(* CoDeSys 2.3.9.42 project: Revers privod_96.pro *)
(* Libraries: STANDARD.LIB 4.10.05 11:14:46, IECSFC.LIB 13.4.06 15:51:28, ANALYZATION.LIB 5.10.99 09:05:06 *)

(* Global variable list: Global_Variables *)
VAR_GLOBAL
	KM1, KM2:BOOL;
END_VAR

(* POU PLC_PRG, ST *)
PROGRAM PLC_PRG
VAR
	posy: INT;
END_VAR
Control();
Puskatel();

IF KM1 THEN
posy:=posy-1;
END_IF

IF KM2 THEN
posy:=posy+1;
END_IF
END_PROGRAM

(* POU Control, LD *)
PROGRAM Control
VAR
	S0: BOOL;
	SI: BOOL;
	SD: BOOL;
END_VAR
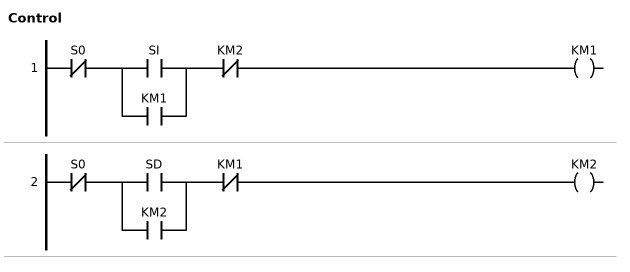
_LD_ (* Ladder Diagram *)
NETWORK 1
	[/S0] - { [SI] | [KM1] } - [/KM2] --- (KM1)
NETWORK 2
	[/S0] - { [SD] | [KM2] } - [/KM1] --- (KM2)
_END_LD_
(* the same logic as Structured Text *)
(* Network 1 *)
KM1 := NOT S0 AND (SI OR KM1) AND NOT KM2;
(* Network 2 *)
KM2 := NOT S0 AND (SD OR KM2) AND NOT KM1;
END_PROGRAM

(* POU Puskatel, LD *)
PROGRAM Puskatel
VAR
	S01: BOOL;
	Start: BOOL;
	KM_1: BOOL;
	Stop: BOOL;
END_VAR
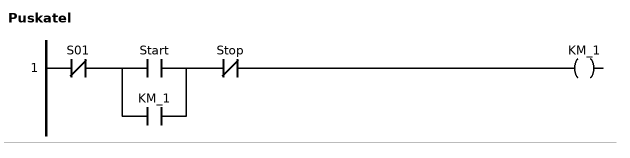
_LD_ (* Ladder Diagram *)
NETWORK 1
	[/S01] - { [Start] | [KM_1] } - [/Stop] --- (KM_1)
_END_LD_
(* the same logic as Structured Text *)
(* Network 1 *)
KM_1 := NOT S01 AND (Start OR KM_1) AND NOT Stop;
END_PROGRAM

(* Visualisation visual
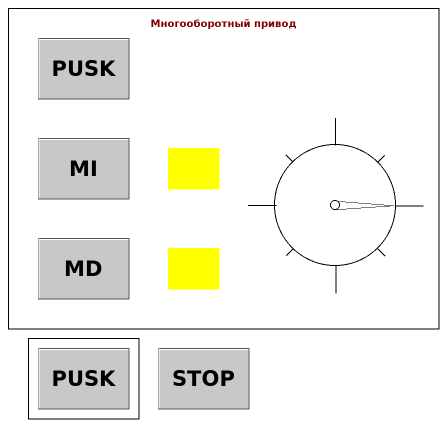
rectangle at (40,350)-(151,431): alarm colour if Puskatel.KM_1
rounded rectangle at (180,160)-(231,201): alarm colour if .KM1
rounded rectangle at (180,260)-(231,301): alarm colour if .KM2
button at (50,50)-(141,111): text "PUSK"; taps Control.S0
rectangle at (140,10)-(331,61): text "Многооборотный привод"
button at (50,150)-(141,211): text "MI"; taps Control.SI
button at (50,250)-(141,311): text "MD"; taps Control.SD
button at (50,360)-(141,421): text "PUSK"; taps Puskatel.Start
button at (170,360)-(261,421): text "STOP"; taps Puskatel.Stop
group at (260,130)-(435,305)
  polygon at (87,83)-(145,91): angle ((PLC_PRG.posy * 1.0)-180) * 1
12 more shapes without text or variables
*)
